% RSLogix 500 project PROJECT2_DIGITAL_FILLING_STATION.RSS, saved by version 8.30.00.16 %
PROJECT "UNTITLED"    % processor: Bul.1763 MicroLogix 1100 Series B %

PROGRAM FILES
  LAD 2   3 rungs
  LAD 3 "IO"  9 rungs
  LAD 4 "CONTROL"  5 rungs

DATA FILES
  O0 OUTPUT  4 elements
  I1 INPUT  6 elements
  S2 STATUS  66 elements
  B3 BINARY  1 elements
  T4 TIMER  1 elements
  C5 COUNTER  1 elements
  R6 CONTROL  1 elements
  N7 INTEGER  1 elements
  F8 FLOAT  1 elements

LADDER 2
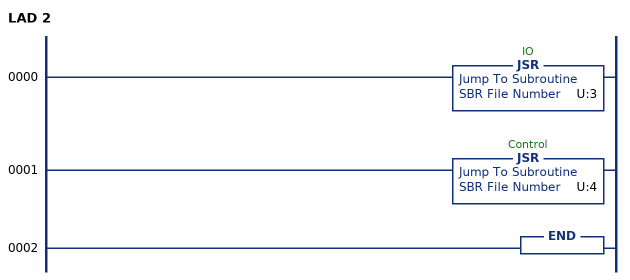
% Rung: 0 %
SOR JSR U:3 EOR
%   U:3  "IO" %
% Rung: 1 %
SOR JSR U:4 EOR
%   U:4  "Control" %
% Rung: 2 %
SOR END EOR

LADDER 3 "IO"
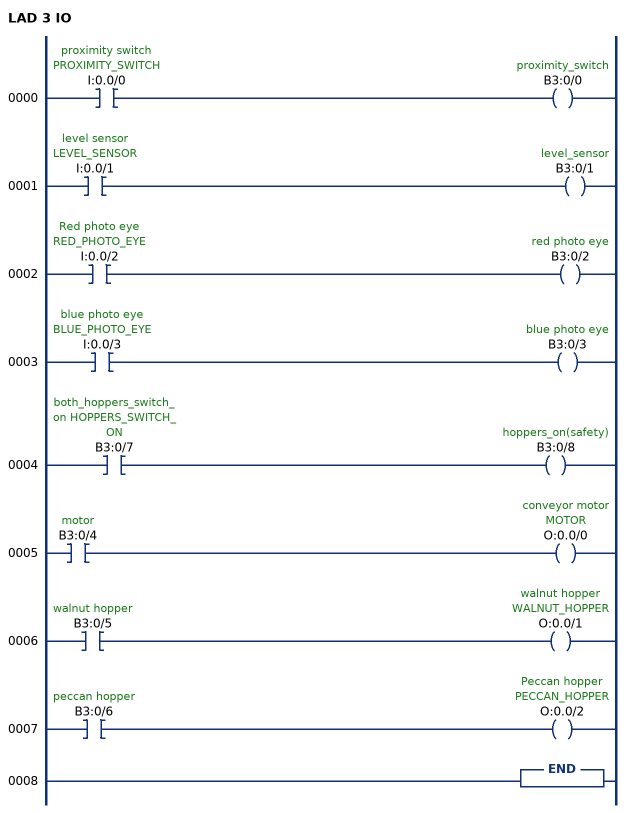
% Rung: 0 %
SOR XIC I:0.0/0 OTE B3:0/0 EOR
%   I:0.0/0  PROXIMITY_SWITCH  "proximity switch" %
%   B3:0/0  "proximity_switch" %
% Rung: 1 %
SOR XIC I:0.0/1 OTE B3:0/1 EOR
%   I:0.0/1  LEVEL_SENSOR  "level sensor" %
%   B3:0/1  "level_sensor" %
% Rung: 2 %
SOR XIC I:0.0/2 OTE B3:0/2 EOR
%   I:0.0/2  RED_PHOTO_EYE  "Red photo eye" %
%   B3:0/2  "red photo eye" %
% Rung: 3 %
SOR XIC I:0.0/3 OTE B3:0/3 EOR
%   I:0.0/3  BLUE_PHOTO_EYE  "blue photo eye" %
%   B3:0/3  "blue photo eye" %
% Rung: 4 %
SOR XIC B3:0/7 OTE B3:0/8 EOR
%   B3:0/7  HOPPERS_SWITCH_ON  "both_hoppers_switch_ on" %
%   B3:0/8  "hoppers_on(safety)" %
% Rung: 5 %
SOR XIC B3:0/4 OTE O:0.0/0 EOR
%   B3:0/4  "motor" %
%   O:0.0/0  MOTOR  "conveyor motor" %
% Rung: 6 %
SOR XIC B3:0/5 OTE O:0.0/1 EOR
%   B3:0/5  "walnut hopper" %
%   O:0.0/1  WALNUT_HOPPER  "walnut hopper" %
% Rung: 7 %
SOR XIC B3:0/6 OTE O:0.0/2 EOR
%   B3:0/6  "peccan hopper" %
%   O:0.0/2  PECCAN_HOPPER  "Peccan hopper" %
% Rung: 8 %
SOR END EOR

LADDER 4 "CONTROL"
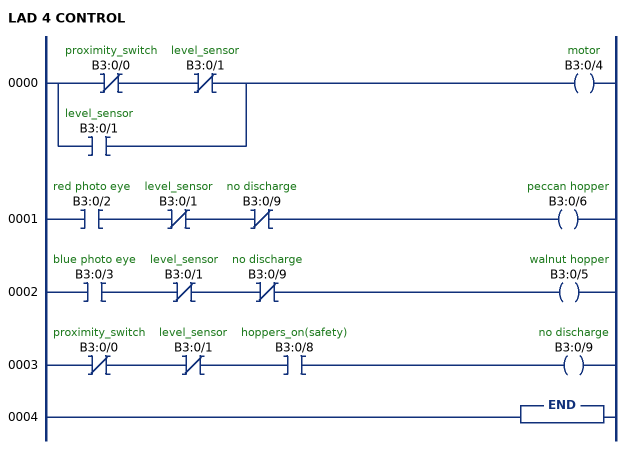
% Rung: 0 %
SOR BST XIO B3:0/0 XIO B3:0/1 NXB XIC B3:0/1 BND OTE B3:0/4 EOR
%   B3:0/0  "proximity_switch" %
%   B3:0/1  "level_sensor" %
%   B3:0/4  "motor" %
% Rung: 1 %
SOR XIC B3:0/2 XIO B3:0/1 XIO B3:0/9 OTE B3:0/6 EOR
%   B3:0/2  "red photo eye" %
%   B3:0/1  "level_sensor" %
%   B3:0/9  "no discharge" %
%   B3:0/6  "peccan hopper" %
% Rung: 2 %
SOR XIC B3:0/3 XIO B3:0/1 XIO B3:0/9 OTE B3:0/5 EOR
%   B3:0/3  "blue photo eye" %
%   B3:0/1  "level_sensor" %
%   B3:0/9  "no discharge" %
%   B3:0/5  "walnut hopper" %
% Rung: 3 %
SOR XIO B3:0/0 XIO B3:0/1 XIC B3:0/8 OTE B3:0/9 EOR
%   B3:0/0  "proximity_switch" %
%   B3:0/1  "level_sensor" %
%   B3:0/8  "hoppers_on(safety)" %
%   B3:0/9  "no discharge" %
% Rung: 4 %
SOR END EOR

OTHER DOCUMENTED ADDRESSES
  B3:0/10  "simulataneous_hopper s_toggle_off"
